Staubli VAL3: HIT_YD.pjx

--- HIT_YD.pjx ---
Parameters version=s7.6.2 stackSize=5000 millimeterUnit=true
Program file=ClientGet.pgx
Program file=ClientSend.pgx
Program file=OMAC_Abort.pgx
Program file=OMAC_Hold.pgx
Program file=OMAC_Main.pgx
Program file=OMAC_Reset.pgx
Program file=OMAC_Start.pgx
Program file=OMAC_Stop.pgx
Program file=OMAC_Unhold.pgx
Program file=blow.pgx
Program file=bypassPick.pgx
Program file=cellManager.pgx
Program file=getToolStatus.pgx
Program file=goHome.pgx
Program file=init.pgx
Program file=initTracking.pgx
Program file=isInSafetyArea.pgx
Program file=modbusGet.pgx
Program file=modbusSet.pgx
Program file=overflowPick.pgx
Program file=Place.pgx
Program file=productionCycle.pgx
Program file=robot2PLC.pgx
Program file=sRobot2fRobot.pgx
Program file=send2NextRob.pgx
Program file=setAlarm.pgx
Program file=setConvSpeed.pgx
Program file=start.pgx
Program file=stop.pgx
Program file=trackErr_init.pgx
Program file=trackingPick.pgx
Program file=transferQueue.pgx
Data file=HIT_YD.dtx
Library alias=mot path=Disk://Tracking/Motion/Motion.pjx autoload=true password=
Type name=object path=Disk://Tracking/Templates/object/object.pjx

--- HIT_YD.dtx ---
aio aConvSpeed = {link=ModbusSrv-0\Modbus-Word\ao[3]}
aio aPlcCmd = {link=ModbusSrv-0\Modbus-Word\ai[0]}
aio aRbAlarm = {link=ModbusSrv-0\Modbus-Word\ao[0]}
aio aRbStatus = {link=ModbusSrv-0\Modbus-Word\ao[1]}
bool _bConvExist = true
bool _bEndCycle
bool _bIsPicking
bool _bIsPlacing
bool _bMutexCnvQueue = true
bool _bPartInTool
bool _bSentToHome = true
bool bIsPermitPlace = true
bool bIsStartPlace = true
bool bLockPage
bool bPickDetection
bool bSetConvSpeed
bool bTransferData
dio dAlarm[8]
  [0] = {link=ModbusSrv-0\Modbus-Bit\do[8]}
  [1] = {link=ModbusSrv-0\Modbus-Bit\do[9]}
  [2] = {link=ModbusSrv-0\Modbus-Bit\do[10]}
  [3] = {link=ModbusSrv-0\Modbus-Bit\do[11]}
  [4] = {link=ModbusSrv-0\Modbus-Bit\do[12]}
  [5] = {link=ModbusSrv-0\Modbus-Bit\do[13]}
  [6] = {link=ModbusSrv-0\Modbus-Bit\do[14]}
  [7] = {link=ModbusSrv-0\Modbus-Bit\do[15]}
dio dBlow = {link=BasicIO-1\%Q5}
dio dControlVacuum[4]
  [0] = {link=BasicIO-1\%Q7}
  [1] = {link=BasicIO-1\%Q6}
  [2] = {link=BasicIO-1\%Q5}
  [3] = {link=BasicIO-1\%Q4}
dio dPartInTool = {link=fIn0}
dio dPermitPlace[4]
  [0] = {link=ModbusSrv-0\Modbus-Bit\di[3]}
  [1] = {link=ModbusSrv-0\Modbus-Bit\di[2]}
  [2] = {link=ModbusSrv-0\Modbus-Bit\di[1]}
  [3] = {link=ModbusSrv-0\Modbus-Bit\di[0]}
dio dPlaceDone[4]
  [0] = {link=ModbusSrv-0\Modbus-Bit\do[3]}
  [1] = {link=ModbusSrv-0\Modbus-Bit\do[2]}
  [2] = {link=ModbusSrv-0\Modbus-Bit\do[1]}
  [3] = {link=ModbusSrv-0\Modbus-Bit\do[0]}
dio dStartControl[4]
  [0] = {link=ModbusSrv-0\Modbus-Bit\di[4]}
  [1] = {link=ModbusSrv-0\Modbus-Bit\di[5]}
  [2] = {link=ModbusSrv-0\Modbus-Bit\di[6]}
  [3] = {link=ModbusSrv-0\Modbus-Bit\di[7]}
dio dStartState[4]
  [0] = {link=ModbusSrv-0\Modbus-Bit\do[4]}
  [1] = {link=ModbusSrv-0\Modbus-Bit\do[5]}
  [2] = {link=ModbusSrv-0\Modbus-Bit\do[6]}
  [3] = {link=ModbusSrv-0\Modbus-Bit\do[7]}
dio dVacuum = {link=BasicIO-1\%Q4}
frame fConveyor = {x=690.465999, y=-334.533545, z=-72.519533, rx=0.736674, ry=-0.299775, rz=179.886741, fatherId=world[0]}
frame fDetection = {x=319.933347, y=-456.969728, z=-77.119399, rx=1.134288, ry=-0.307561, rz=179.705392, fatherId=world[0]}
jointRs jDropPart = {j1=-61.262813, j2=45.342289, j3=74.332986, j4=152.342331}
jointRs jHome = {j1=-61.262813, j2=45.342289, j3=74.332986, j4=152.342331}
jointRs jPark = {j1=-61.262813, j2=45.342289, j3=74.332986, j4=152.342331}
mdesc _mLoad = {accel=64, vel=80, decel=64, leave=30, reach=30}
mdesc mLoad = {accel=64, vel=80, decel=64, leave=30, reach=30}
mdesc mNomSpeed = {accel=144, vel=120, decel=144, leave=20, reach=20}
mdesc mPickDown = {accel=169, vel=130, decel=169, blend=off, leave=30, reach=30}
mdesc mPickup = {accel=144, vel=120, decel=144}
mdesc mPlaceDown = {accel=144, vel=120, decel=144, blend=off, leave=15, reach=15}
mdesc mPlaceUp = {accel=169, vel=130, decel=169, blend=cartesian, leave=30, reach=30}
mdesc mSlow = {accel=1, vel=10, decel=1, leave=10, reach=10}
mdesc mUnload = {accel=121, vel=120, decel=121, leave=40, reach=40}
num _nBlowDelay
num _nCntBypassed
num _nCntPartsDone[2]
  [0] = 13306
  [1] = 13306
num _nCntTransfered = 8
num _nConvSpd = 491.491944
num _nCycleTime[10]
  [0] = 0.964
  [1] = 2.051
  [2] = 0.756
  [3] = 4.461
  [4] = 0.846
  [5] = 4.253
  [6] = 0.92
  [7] = 8.599
  [8] = 0.993
  [9] = 2.124
num _nCycleTimeIndx
num _nID = -1
num _nLastStateCMD
num _nOmacStat = 3
num _nPartID = 1
num _nPlaceCurItem[2]
num _nPullIndexTQ
num _nPushIndexTQ
num _nStateCMD
num _nTimer = 7404.541
num _nTrackErr = 46
num nBlowID = 0.5
num nBypass
num nLoadRatio[4]
  [0] = 1
  [1] = 0.85
  [2] = 0.7
  [3] = 0.7
num nNomConvSpeed = 100
num nPartHeight = 8
num nPickAppro = 60
num nPlaceAppro = 50
num nPlaceCycleNum = 1
public num nPlaceNum = 1
num nSafeMaxX = 850
num nSafeMaxY = 850
num nSafeMinX = -850
num nSafeMinY = -850
num nTestData[5]
  [0] = 1
  [1] = 8
  [3] = -7
num nVacuumID = 0.2
num nWaitDist2Up4BP = -150
num nWaitDistToDown = 50
num nWaitDistToUp[1 3]
  [0,0] = -50
  [0,1] = 200
  [0,2] = 400
num nWaitDistX = -150
object _oTransferQueue[1 100]
  [0,0]
    num nID = -1
    num nLatchedValue
    trsf trTrsf
  [0,1]
    num nID = -1
    num nLatchedValue
    trsf trTrsf
  [0,2]
    num nID = -1
    num nLatchedValue
    trsf trTrsf
  [0,3]
    num nID = -1
    num nLatchedValue
    trsf trTrsf
  [0,4]
    num nID = -1
    num nLatchedValue
    trsf trTrsf
  [0,5]
    num nID = -1
    num nLatchedValue
    trsf trTrsf
  [0,6]
    num nID = -1
    num nLatchedValue
    trsf trTrsf
  [0,7]
    num nID = -1
    num nLatchedValue
    trsf trTrsf
  [0,8]
    num nID = -1
    num nLatchedValue
    trsf trTrsf
  [0,9]
    num nID = -1
    num nLatchedValue
    trsf trTrsf
  [0,10]
    num nID = -1
    num nLatchedValue
    trsf trTrsf
  [0,11]
    num nID = -1
    num nLatchedValue
    trsf trTrsf
  [0,12]
    num nID = -1
    num nLatchedValue
    trsf trTrsf
  [0,13]
    num nID = -1
    num nLatchedValue
    trsf trTrsf
  [0,14]
    num nID = -1
    num nLatchedValue
    trsf trTrsf
  [0,15]
    num nID = -1
    num nLatchedValue
    trsf trTrsf
  [0,16]
    num nID = -1
    num nLatchedValue
    trsf trTrsf
  [0,17]
    num nID = -1
    num nLatchedValue
    trsf trTrsf
  [0,18]
    num nID = -1
    num nLatchedValue
    trsf trTrsf
  [0,19]
    num nID = -1
    num nLatchedValue
    trsf trTrsf
  [0,20]
    num nID = -1
    num nLatchedValue
    trsf trTrsf
  [0,21]
    num nID = -1
    num nLatchedValue
    trsf trTrsf
  [0,22]
    num nID = -1
    num nLatchedValue
    trsf trTrsf
  [0,23]
    num nID = -1
    num nLatchedValue
    trsf trTrsf
  [0,24]
    num nID = -1
    num nLatchedValue
    trsf trTrsf
  [0,25]
    num nID = -1
    num nLatchedValue
    trsf trTrsf
  [0,26]
    num nID = -1
    num nLatchedValue
    trsf trTrsf
  [0,27]
    num nID = -1
    num nLatchedValue
    trsf trTrsf
  [0,28]
    num nID = -1
    num nLatchedValue
    trsf trTrsf
  [0,29]
    num nID = -1
    num nLatchedValue
    trsf trTrsf
  [0,30]
    num nID = -1
    num nLatchedValue
    trsf trTrsf
  [0,31]
    num nID = -1
    num nLatchedValue
    trsf trTrsf
  [0,32]
    num nID = -1
    num nLatchedValue
    trsf trTrsf
  [0,33]
    num nID = -1
    num nLatchedValue
    trsf trTrsf
  [0,34]
    num nID = -1
    num nLatchedValue
    trsf trTrsf
  [0,35]
    num nID = -1
    num nLatchedValue
    trsf trTrsf
  [0,36]
    num nID = -1
    num nLatchedValue
    trsf trTrsf
  [0,37]
    num nID = -1
    num nLatchedValue
    trsf trTrsf
  [0,38]
    num nID = -1
    num nLatchedValue
    trsf trTrsf
  [0,39]
    num nID = -1
    num nLatchedValue
    trsf trTrsf
  [0,40]
    num nID = -1
    num nLatchedValue
    trsf trTrsf
  [0,41]
    num nID = -1
    num nLatchedValue
    trsf trTrsf
  [0,42]
    num nID = -1
    num nLatchedValue
    trsf trTrsf
  [0,43]
    num nID = -1
    num nLatchedValue
    trsf trTrsf
  [0,44]
    num nID = -1
    num nLatchedValue
    trsf trTrsf
  [0,45]
    num nID = -1
    num nLatchedValue
    trsf trTrsf
  [0,46]
    num nID = -1
    num nLatchedValue
    trsf trTrsf
  [0,47]
    num nID = -1
    num nLatchedValue
    trsf trTrsf
  [0,48]
    num nID = -1
    num nLatchedValue
    trsf trTrsf
  [0,49]
    num nID = -1
    num nLatchedValue
    trsf trTrsf
  [0,50]
    num nID = -1
    num nLatchedValue
    trsf trTrsf
  [0,51]
    num nID = -1
    num nLatchedValue
    trsf trTrsf
  [0,52]
    num nID = -1
    num nLatchedValue
    trsf trTrsf
  [0,53]
    num nID = -1
    num nLatchedValue
    trsf trTrsf
  [0,54]
    num nID = -1
    num nLatchedValue
    trsf trTrsf
  [0,55]
    num nID = -1
    num nLatchedValue
    trsf trTrsf
  [0,56]
    num nID = -1
    num nLatchedValue
    trsf trTrsf
  [0,57]
    num nID = -1
    num nLatchedValue
    trsf trTrsf
  [0,58]
    num nID = -1
    num nLatchedValue
    trsf trTrsf
  [0,59]
    num nID = -1
    num nLatchedValue
    trsf trTrsf
  [0,60]
    num nID = -1
    num nLatchedValue
    trsf trTrsf
  [0,61]
    num nID = -1
    num nLatchedValue
    trsf trTrsf
  [0,62]
    num nID = -1
    num nLatchedValue
    trsf trTrsf
  [0,63]
    num nID = -1
    num nLatchedValue
    trsf trTrsf
  [0,64]
    num nID = -1
    num nLatchedValue
    trsf trTrsf
  [0,65]
    num nID = -1
    num nLatchedValue
    trsf trTrsf
  [0,66]
    num nID = -1
    num nLatchedValue
    trsf trTrsf
  [0,67]
    num nID = -1
    num nLatchedValue
    trsf trTrsf
  [0,68]
    num nID = -1
    num nLatchedValue
    trsf trTrsf
  [0,69]
    num nID = -1
    num nLatchedValue
    trsf trTrsf
  [0,70]
    num nID = -1
    num nLatchedValue
    trsf trTrsf
  [0,71]
    num nID = -1
    num nLatchedValue
    trsf trTrsf
  [0,72]
    num nID = -1
    num nLatchedValue
    trsf trTrsf
  [0,73]
    num nID = -1
    num nLatchedValue
    trsf trTrsf
  [0,74]
    num nID = -1
    num nLatchedValue
    trsf trTrsf
  [0,75]
    num nID = -1
    num nLatchedValue
    trsf trTrsf
  [0,76]
    num nID = -1
    num nLatchedValue
    trsf trTrsf
  [0,77]
    num nID = -1
    num nLatchedValue
    trsf trTrsf
  [0,78]
    num nID = -1
    num nLatchedValue
    trsf trTrsf
  [0,79]
    num nID = -1
    num nLatchedValue
    trsf trTrsf
  [0,80]
    num nID = -1
    num nLatchedValue
    trsf trTrsf
  [0,81]
    num nID = -1
    num nLatchedValue
    trsf trTrsf
  [0,82]
    num nID = -1
    num nLatchedValue
    trsf trTrsf
  [0,83]
    num nID = -1
    num nLatchedValue
    trsf trTrsf
  [0,84]
    num nID = -1
    num nLatchedValue
    trsf trTrsf
  [0,85]
    num nID = -1
    num nLatchedValue
    trsf trTrsf
  [0,86]
    num nID = -1
    num nLatchedValue
    trsf trTrsf
  [0,87]
    num nID = -1
    num nLatchedValue
    trsf trTrsf
  [0,88]
    num nID = -1
    num nLatchedValue
    trsf trTrsf
  [0,89]
    num nID = -1
    num nLatchedValue
    trsf trTrsf
  [0,90]
    num nID = -1
    num nLatchedValue
    trsf trTrsf
  [0,91]
    num nID = -1
    num nLatchedValue
    trsf trTrsf
  [0,92]
    num nID = -1
    num nLatchedValue
    trsf trTrsf
  [0,93]
    num nID = -1
    num nLatchedValue
    trsf trTrsf
  [0,94]
    num nID = -1
    num nLatchedValue
    trsf trTrsf
  [0,95]
    num nID = -1
    num nLatchedValue
    trsf trTrsf
  [0,96]
    num nID = -1
    num nLatchedValue
    trsf trTrsf
  [0,97]
    num nID = -1
    num nLatchedValue
    trsf trTrsf
  [0,98]
    num nID = -1
    num nLatchedValue
    trsf trTrsf
  [0,99]
    num nID = -1
    num nLatchedValue
    trsf trTrsf
pointRs pPick = {shoulder=righty, fatherId=fDetection[0]}
pointRs pPlace[4]
  [0] = {x=752.590073, y=-120.83, z=-69.15, rx=180, rz=95.410382, shoulder=righty, fatherId=world[0]}
  [1] = {x=614.985623, y=-120.83, z=-69.15, rx=180, rz=95.41037, shoulder=righty, fatherId=world[0]}
  [2] = {x=479.250185, y=-120.83, z=-69.15, rx=180, rz=95.410122, shoulder=righty, fatherId=world[0]}
  [3] = {x=345.150595, y=-120.83, z=-69.15, rx=180, rz=95.409269, shoulder=righty, fatherId=world[0]}
sio sClient = {link=Socket\StlClient}
sio skToRobot = {link=Socket\toRobot_sk1}
string _sCycleStatus = "Waiting for part to pick"
string sConveyorList = "cvIn"
string sSecondRStatus = "8"
tool tGripper = {z=75, rz=-128, fatherId=flange[0], ioLink=valve1}
public trsf trTrsfPlace[4]
  [1] = {x=140}
  [2] = {x=280}
  [3] = {x=420}

--- cellManager.pgx ---
program cellManager()
  local joint l_jHere
  local num l_nConvSpeedOld
  local num l_nErr
  local num l_nI
begin
  // This program is the cell manager, it manage:
  //  -  Variable initializing
  //  -  Launch Tracking
  //  -  Arm Power
  //  -  Robot home position
  //  -  Launch user’s tasks, kills and re-launch user’s task in case of tracking error
  //  -  Displays cycle times and counters.
  //
  // Input parameters
  //  None            :
  //
  // Output parameters
  //  None            :
  //
  //----------------------------------------------------------------
  //

  //  //Launch queue transfer tasks
  //  if _bTransferData[0]
  //    taskCreate "TransferQueue1",100,transferQueue(0)
  //  endIf
  //  // Task to remove picking positions that have pass the downstream limit while the robot is placing a part.
  //  taskCreate "overflowPick",100,overflowPick()

  // Task for production cycle
  if taskStatus("productionCycle")>=0
    taskKill("productionCycle")
  endIf
  wait(taskStatus("productionCycle")<0)
  taskCreate "productionCycle",100,productionCycle()


  // Task to set the blow on the tool for a defined period of time
  if taskStatus("blow")>=0
    taskKill("blow")
  endIf
  wait(taskStatus("blow")<0)
  taskCreate "blow",100,blow()
  wait(taskStatus("blow")==1)
  //
  if taskStatus("sRobot2fRobot")>=0
    taskKill("sRobot2fRobot")
  endIf
  wait(taskStatus("sRobot2fRobot")<0)
  taskCreate "sRobot2fRobot",100,sRobot2fRobot()
  //
  if taskStatus("robot2PLC")>=0
    taskKill("robot2PLC")
  endIf
  wait(taskStatus("robot2PLC")<0)
  taskCreate "robot2PLC",100,robot2PLC()

  //OMAC进程:Running
  _nOmacStat=3

  //
  //  //Init conveyor speed
  //  call setConvSpeed(0,nNomConvSpeed[0])
  //  l_nConvSpeedOld[0]=nNomConvSpeed[0]
  //
  // Main loop
  do
    // Enable Power
    if isPowered()==false and esStatus()!=2
      if _nOmacStat==3
        enablePower()
        delay(0.5)
      endIf
    endIf
    //
    // Set conveyor speed to the nominal value if the conveyor speed is not controlled by the tasks
    //  overflowPick and overflowPlace
    if bSetConvSpeed[0]
      l_nConvSpeedOld[0]=0
    else
      if l_nConvSpeedOld[0]!=nNomConvSpeed[0]
        call setConvSpeed(0,nNomConvSpeed[0])
        l_nConvSpeedOld[0]=nNomConvSpeed[0]
      endIf
    endIf

    if _nOmacStat==3
      //task TransferQueue1 error management,auto recover
      if bTransferData[0]
        if taskStatus("TransferQueue1")!=1
          logMsg("TransferQueue1任务错误")
          taskKill("TransferQueue1")
          wait(taskStatus("TransferQueue1")==-1)
          taskCreate "TransferQueue1",100,transferQueue(0)
          wait(taskStatus("TransferQueue1")==1)
          logMsg("TransferQueue1自动恢复")
        endIf
      endIf
      //task TransferQueue1 error management,auto recover
      if taskStatus("overflowPick")!=1
        logMsg("overflowPick任务错误")
        taskKill("overflowPick")
        wait(taskStatus("overflowPick")==-1)
        taskCreate "overflowPick",100,overflowPick()
        wait(taskStatus("overflowPick")==1)
        logMsg("overflowPick自动恢复")
      endIf
      // Tracking error management
      if isSettled()==true and $trackingState()==-1
        if _nOmacStat==3
          if _bIsPicking==true
            logMsg("抓取时跟踪错误")
          endIf
          if _bIsPlacing==true
            logMsg("放件时运动错误")
          endIf
          //记录跟踪错误次数
          _nTrackErr=_nTrackErr+1
          stopMove()
          resetMotion()
          call trackErr_init()
          autoConnectMove(true)
          l_jHere=herej()
          l_jHere.j3=jHome.j3
          movej(l_jHere,tGripper,mNomSpeed)
          movej(jHome,tGripper,mNomSpeed)
          _bSentToHome=true
          //          //Launch queue transfer tasks
          //          if _bTransferData[0]
          //            taskCreate "TransferQueue1",100,transferQueue(0)
          //          endIf
          //          // Task to remove picking positions that have pass the downstream limit while the robot is placing a part.
          //          taskCreate "overflowPick",100,overflowPick()
          // Task for production cycle

          if taskStatus("productionCycle")>=0
            taskKill("productionCycle")
          endIf
          wait(taskStatus("productionCycle")<0)
          taskCreate "productionCycle",100,productionCycle()
          wait(taskStatus("productionCycle")==1)
        endIf
      endIf
    endIf
    //
    //show cv speed
    if _bConvExist
      call mot:getConvSpeed(0,_nConvSpd,l_nErr)
      gotoxy(0,0)
      put("                    ")
      gotoxy(0,0)
      put("传送带速度："+toString("",_nConvSpd)+" mm/s")
    endIf


    delay(0)
  until false
end

--- init.pgx ---
program init()
  local num l_nI
  local num l_nJ
begin
  // This program initialize all variables
  //
  // Input parameters
  //  None            :
  //
  // Output parameters
  //  None            :
  //
  //----------------------------------------------------------------
  //
  //che add
  nPlaceNum=0
  nPlaceCycleNum=0
  bIsPermitPlace=true
  sSecondRStatus=""
  // Booleans
  _bSentToHome=false
  _bMutexCnvQueue[0]=false
  _bIsPicking=false
  _bIsPlacing=false
  _bConvExist=false
  _bEndCycle=false
  //

  //
  // Numerical
  _nBlowDelay=0
  _nID[0]=-1
  _nCntBypassed[0]=nBypass[0]
  _nCntTransfered[0]=0

  _nPushIndexTQ[0]=0
  _nPullIndexTQ[0]=0
  _nTimer=0

  resize(_nCycleTime,1,10)
  for _nCycleTimeIndx=0 to size(_nCycleTime)-1
    _nCycleTime[_nCycleTimeIndx]=0
  endFor
  _nCycleTimeIndx=0

  //dio
  dPlaceDone[0]=false
  dPlaceDone[1]=false
  dPlaceDone[2]=false
  dPlaceDone[3]=false

  // aio
  aioSet(aRbAlarm,0)
  //call setAlarm(0)

  //
  // Points
  pPick.trsf={0,0,0,0,0,0}

  //

  //
  // Transfer Queues
  for l_nI=0 to size(_oTransferQueue,2)-1
    _oTransferQueue[0,l_nI].nID=-1
    _oTransferQueue[0,l_nI].trTrsf={0,0,0,0,0,0}
    _oTransferQueue[0,l_nI].nLatchedValue=0
  endFor
  //
  // Strings
  _sCycleStatus=""
end

--- isInSafetyArea.pgx ---
program isInSafetyArea()
  local jointRs l_jHere
  local pointRs l_pCurrent
begin
  do
    l_pCurrent=here(flange,world)
    //**************************************************//
    //******** 用来判断机器人是否在安全工作空间 ********//
    //**************************************************//
    if (l_pCurrent.trsf.y>=nSafeMaxY or l_pCurrent.trsf.y<=nSafeMinY or l_pCurrent.trsf.x>=nSafeMaxX or l_pCurrent.trsf.x<=nSafeMinX) and _nOmacStat==3
      aioSet(aRbAlarm,10)
      call setAlarm(7)
      popUpMsg("机器人超出安全工作空间！")
      logMsg("机器人超出安全工作空间！")
      call OMAC_Abort()
    endIf
    delay(0)
  until false
end

--- OMAC_Main.pgx ---
program OMAC_Main()
begin
  //  _nOmacStat
  //1-Ready
  //2-Starting
  //3-Running
  //4-Resetting
  //5-Holding
  //6-Held
  //7-Un-Holding
  //8-Stopping
  //9-Stopped
  //10-Aborting


  // _nStateCmd
  //1-Start
  //2-Stop
  //3-Reset
  //4-Hold
  //10-Abort

  //机器人状态
  _nOmacStat=9

  _nLastStateCMD=0
  //OMAC_init
  call init()
  do
    switch _nOmacStat
      //复位信号
      case 1
        call modbusSet(3)
      break
      //运行信号
      case 3
        call modbusSet(1)
      break
      //准备信号
      case 4
        call modbusSet(2)
      break
      //停止信号
      case 9
        call modbusSet(2)
      break
    endSwitch
    //机器人状态输出
    //aioSet(aRbStatus,_nOmacStat)
    //根据上位机按钮转换为指令num
    //10-Abort
    if esStatus()==2
      _nStateCMD=10
    else
      call modbusGet(_nStateCMD)

      //_nStateCMD=aioGet(aPlcCmd)
    endIf

    //根据指令num，触发相应动作
    if _nStateCMD!=_nLastStateCMD
      switch _nStateCMD
        //Reset
        case 3
          //确认当前OMAC进程为stopped
          if _nOmacStat==9

            if taskStatus("Reset")>=0
              taskKill("Reset")
            endIf
            wait(taskStatus("Reset")<0)
            taskCreate "Reset",100,OMAC_Reset()

          endIf
        break

        //Start
        case 1
          //确认当前OMAC进程为Ready
          if _nOmacStat==1

            if taskStatus("Start")>=0
              taskKill("Start")
            endIf
            wait(taskStatus("Start")<0)
            taskCreate "Start",100,OMAC_Start()


          elseIf _nOmacStat==6
            //确认当前OMAC进程为Held

            if taskStatus("Unhold")>=0
              taskKill("Unhold")
            endIf
            wait(taskStatus("Unhold")<0)
            taskCreate "Unhold",100,OMAC_Unhold()

          endIf
        break
        //Hold
        case 4
          //确认当前OMAC进程为running
          if _nOmacStat==3

            if taskStatus("Hold")>=0
              taskKill("Hold")
            endIf
            wait(taskStatus("Hold")<0)
            taskCreate "Hold",100,OMAC_Hold()

          endIf
        break

        //Unhold
        case 7

        break

        //Stop
        case 2
          //确认当前OMAC进程不是停止
          if _nOmacStat!=9
            if taskStatus("Stop")>=0
              taskKill("Stop")
            endIf
            wait(taskStatus("Stop")<0)
            taskCreate "Stop",100,OMAC_Stop()
          endIf
        break

        //Abort
        case 10
          // //确认当前OMAC进程不是停止
          if _nOmacStat!=9
            if taskStatus("Abort")>=0
              taskKill("Abort")
            endIf
            wait(taskStatus("Abort")<0)
            taskCreate "Abort",100,OMAC_Abort()
          endIf
        break

      endSwitch
    endIf
    //记录上次指令
    _nLastStateCMD=_nStateCMD
    delay(0)
  until false


end

--- OMAC_Stop.pgx ---
program OMAC_Stop()
  local joint l_jHere
  local string l_sToolStatus
begin

  //OMAC进程:Stopping
  _nOmacStat=8
  logMsg("上位机手动操作：停止")
  stopMove()
  resetMotion()
  //
  // Stop task

  taskKill("cellManager")
  taskKill("overflowPick")
  taskKill("productionCycle")
  taskKill("Reset")
  taskKill("Start")
  taskKill("Hold")
  taskKill("Unhold")
  taskKill("Preheat")
  taskKill("openPallet")
  taskKill("changeBox")
  taskKill("convStopCheck")
  taskKill("TransferQueue1")
  taskKill("robot2PLC")
  taskKill("sRobot2fRobot")


  resetMotion()
  while !isPowered()
    enablePower()
    delay(1)
  endWhile
  //
  // Move up axis 3
  l_jHere=herej()
  l_jHere.j3=95
  movej(l_jHere,tGripper,mSlow)
  //
  // Drop the part on the tool
  if bPickDetection==true
    call getToolStatus(l_sToolStatus)
  endIf
  if l_sToolStatus=="PartInTool" or !bPickDetection
    movej(jDropPart,tGripper,mSlow)
    waitEndMove()
    dVacuum=false
  else
    dVacuum=false
  endIf
  //
  // Go to park position
  movej(jPark,tGripper,mSlow)
  waitEndMove()
  wait(taskStatus("Reset")==-1)
  wait(taskStatus("Start")==-1)
  wait(taskStatus("Hold")==-1)
  wait(taskStatus("Unhold")==-1)
  wait(taskStatus("Preheat")==-1)
  wait(taskStatus("openPallet")==-1)
  wait(taskStatus("changeBox")==-1)
  wait(taskStatus("convStopCheck")==-1)
  wait(taskStatus("cellManager")==-1)
  wait(taskStatus("TransferQueue1")==-1)
  wait(taskStatus("overflowPick")==-1)
  wait(taskStatus("productionCycle")==-1)

  if _bConvExist
    call mot:kill()
    _bConvExist=false
  endIf

  disablePower()
  wait(isPowered()==false)
  //OMAC进程:Stopped
  _nOmacStat=9

  delay(0)
end

--- Place.pgx ---
program place()
  local bool l_bNoError
  local joint l_jAppro
  local num l_nConvNum
  local num l_nError
  local num l_nMoveID
  local num l_nTrackStatus
  local pointRs l_pAppro
  local pointRs l_pPlace
  local string l_sToolStatus
begin
  l_nConvNum=1
  link(l_pPlace,world)
  //che modify start
  if nPlaceNum>3
    nPlaceNum=0
  endIf
  _mLoad=mLoad
  _mLoad.vel=mLoad.vel*nLoadRatio[nPlaceNum]
  _mLoad.accel=mLoad.accel*nLoadRatio[nPlaceNum]*nLoadRatio[nPlaceNum]
  _mLoad.decel=mLoad.decel*nLoadRatio[nPlaceNum]*nLoadRatio[nPlaceNum]
  if nPlaceCycleNum>7
    nPlaceCycleNum=0
  endIf

  //dControlVacuum[nPlaceNum]=false
  l_pPlace=pPlace[nPlaceNum]
  //end
  // Place part
  l_pAppro=appro(l_pPlace,{0,0,-nPlaceAppro,0,0,0})
  l_bNoError=pointToJoint(tGripper,jHome,l_pAppro,l_jAppro)
  call mot:getTrackStatus(l_nTrackStatus)
  if l_nTrackStatus>0
    // Use trackOff if the robot is synchronized
    if l_bNoError
      call mot:trackOffJ(l_jAppro,tGripper,_mLoad,l_nMoveID,l_nError)
    else
      call mot:trackOff(l_pAppro,tGripper,_mLoad,l_nMoveID,l_nError)
    endIf
  else
    // Use movej if the robot is not synchronized
    if l_bNoError
      l_nMoveID=movej(l_jAppro,tGripper,_mLoad)
    else
      l_nMoveID=movej(l_pAppro,tGripper,_mLoad)
    endIf
  endIf
  // wait permit signal
  wait(bIsPermitPlace==true)
  wait(dPermitPlace[nPlaceNum]==true)
  movel(l_pPlace,tGripper,mPlaceDown)
  l_nMoveID=movel(l_pAppro,tGripper,mPlaceUp)
  // check PartInTool if bPickDetection
  if bPickDetection
    //wait(getMoveId()>l_nMoveID-0.8)
    wait(getMoveId()>l_nMoveID+nBlowID-1.1)
    call getToolStatus(l_sToolStatus)
  else
    wait(getMoveId()>l_nMoveID+nBlowID-1.1)
    _bPartInTool=false
  endIf
  //Blow
  wait(getMoveId()>l_nMoveID+nBlowID-1)
  _nBlowDelay=0.15
  // send done signal
  //dPlaceDone[nPlaceNum]=true
  wait(getMoveId()>l_nMoveID+0.1)
  delay(0)
  //dPlaceDone[nPlaceNum]=false
  if l_sToolStatus=="PartInTool" or _bPartInTool==false
    // A part has been placed
    _nCntPartsDone[l_nConvNum]=_nCntPartsDone[l_nConvNum]+1
  endIf
  delay(0)
  //che modify start
  delay(0)

  //sClient=toString("",nPlaceCycleNum)
  nPlaceCycleNum=nPlaceCycleNum+1
  nPlaceNum=nPlaceNum+1
  dPlaceDone[nPlaceNum-1]=true
  //end

end

--- productionCycle.pgx ---
program productionCycle()
  local bool l_bPartDone
  local string l_sToolStatus
begin
  // This program is the main cycle. It pick on part from the input
  // conveyor and places it on an empty cavity on the output conveyor.
  //
  // Input parameters
  //  None            :
  //
  // Output parameters
  //  None            :
  //
  //----------------------------------------------------------------
  //
  // In order to improve cycle time, vacuum is always on, even while
  //  placing a part. To place a part, the blow is activated for a
  //  short period of time when the robot arrives to the place position.
  //
  // Main loop

  call getToolStatus(l_sToolStatus)
  if (!bPickDetection and _bPartInTool==true) or (bPickDetection and l_sToolStatus=="PartInTool")
    call place()
  endIf
  //---------------------------------------------------------------------//
  do
    //Takes control of the Pick conveyor queue.
    setMutex(_bMutexCnvQueue[0])
    do
      call trackingPick(l_bPartDone)
      delay(0)
    until l_bPartDone
    // Release control of the Pick conveyor queue.
    _bMutexCnvQueue[0]=false

    //
    call place()
    //
    delay(0)
  until _bEndCycle
  _bEndCycle=true
  //
end

--- robot2PLC.pgx ---
program robot2PLC()
  local num l_nLocalNum
  local num l_nNextNum
  local num l_ns
begin
  l_nLocalNum=-1
  while true
    //

    wait(dPlaceDone[0]==true or dPlaceDone[1]==true or dPlaceDone[2]==true or dPlaceDone[3]==true)
    //
    l_ns=clock()
    do
      delay(0)
    until clock()-l_ns>0.25

    if (dPlaceDone[0]==true)
      dPlaceDone[0]=false
    elseIf (dPlaceDone[1]==true)
      dPlaceDone[1]=false
    elseIf (dPlaceDone[2]==true)
      dPlaceDone[2]=false
    elseIf (dPlaceDone[3]==true)
      dPlaceDone[3]=false
    else
      dPlaceDone[0]=false
      dPlaceDone[1]=false
      dPlaceDone[2]=false
      dPlaceDone[3]=false
    endIf
    //
    sClient=toString("",nPlaceCycleNum)
    //    if (l_nLocalNum!=nPlaceCycleNum)
    //      //
    //      sClient=toString("",nPlaceCycleNum)
    //      l_nLocalNum=nPlaceCycleNum
    //    endIf

    nTestData[0]=nPlaceCycleNum
    nTestData[1]=asc(sSecondRStatus,0)-48
    nTestData[3]=nTestData[0]-nTestData[1]
  endWhile
end

--- sRobot2fRobot.pgx ---
program sRobot2fRobot()
begin

  //没有ClearBuffer 这个比较难联通
  clearBuffer(sClient)

  //把客户端收到不为空的信息通过服务器传送出去
  while true
    //服务器
    //clearBuffer(sServer)

    call ClientGet(sSecondRStatus)
    //popUpMsg(sFirstRStatus)

    delay(0)
  endWhile

end

--- stop.pgx ---
program stop()
  local joint l_jHere
  local string l_sToolStatus
begin
  //
  l_sToolStatus=""
  //
  cls()
  gotoxy(10,6)
  put("Application Ending")
  //
  stopMove()
  resetMotion()
  disablePower()
  // Stop all tasks
  taskKill("TransferQueue1")
  taskKill("overflowPick")
  taskKill("productionCycle")
  taskKill("blow")
  taskKill("changePallet")
  taskKill("isInSafetyArea")
  taskKill("robot2PLC")
  taskKill("sRobot2fRobot")

  if _bConvExist
    call mot:kill()
  endIf

  //
  // Stop conveyor speed
  call setConvSpeed(0,0)
  //
  // Reset triggers
  //  dioSet(dTrigger,0)
  //
  resetMotion()
  //
  //
  // Move up axis 3
  l_jHere=herej()
  l_jHere.j3=90
  //movej(l_jHere,flange,mSlow)
  //
  // Drop the part on the tool
  if bPickDetection
    call getToolStatus(l_sToolStatus)
  endIf
  if l_sToolStatus=="PartInTool" or !bPickDetection
    //movej(jDropPart,flange,mSlow)
    //waitEndMove()
    dBlow=true
    dVacuum=false
    delay(0.5)
    dBlow=false
  else
    dVacuum=false
    dBlow=false
  endIf
  //
  // Go to park position
  //movej(jPark,flange,mSlow)
  //waitEndMove()
  disablePower()
  //
  cls()
  gotoxy(10,6)
  put("Application Ended")
  //
end

--- trackErr_init.pgx ---
program trackErr_init()
  local num l_nI
begin
  // This program initialize all variables
  //
  // Input parameters
  //  None            :
  //
  // Output parameters
  //  None            :
  //
  //----------------------------------------------------------------
  //
  // Booleans
  _bSentToHome=false
  _bMutexCnvQueue[0]=false
  _bIsPicking=false
  _bIsPlacing=false
  //

  //
  // Numerical
  _nID[0]=-1
  _nCntBypassed[0]=nBypass[0]


  _nPushIndexTQ[0]=0
  _nPullIndexTQ[0]=0
  _nTimer=0

  for _nCycleTimeIndx=0 to 9
    _nCycleTime[_nCycleTimeIndx]=0
  endFor
  _nCycleTimeIndx=0
  //
  // Points
  pPick.trsf={0,0,0,0,0,0}

  //
  // Transfer Queues
  for l_nI=0 to size(_oTransferQueue,2)-1
    _oTransferQueue[0,l_nI].nID=-1
    _oTransferQueue[0,l_nI].trTrsf={0,0,0,0,0,0}
    _oTransferQueue[0,l_nI].nLatchedValue=0
  endFor
  //
  // Strings
  _sCycleStatus=""
end

--- trackingPick.pgx ---
program trackingPick(bool& x_bPartDone (dimensions=1))
  local bool l_bNoError
  local bool l_bSent2WaitPos
  local joint l_jAppro
  local num l_nConvNum
  local num l_nDistToDown
  local num l_nDistToUp
  local num l_nEncLatchVal
  local num l_nError
  local num l_nMoveID
  local num l_nTrackOnID
  local num l_nTrackStatus
  local point l_pAppro
  local string l_sToolStatus
begin
  // This program picks a part from the input conveyor.
  // If there isn’t an object on the conveyor’s queue, the robot
  //  moves to the home position and waits until there is an object
  //  on the conveyor’s queue.
  // If there is an object on the conveyor’s queue but the object is
  //  upstream of the upstream limit, the robot moves above the
  //  conveyor aligned in front of the object and waits until the
  //  object crosses the upstream limit.
  // If the object is in between the upstream and downstream limit,
  //  the robot picks the part.
  // If the object is downstream of the downstream limit, the object
  //  is removed from the conveyor’s queue and the robot is sent to
  //  the home position.
  //
  // Input parameters
  //  None            :
  //
  // Output parameters
  //  x_bPartDone     : A part has been picked
  //
  //----------------------------------------------------------------
  //
  l_nConvNum=0
  x_bPartDone=false
  l_sToolStatus=""
  //
  // If the overflowPick task hasn't already detect the next part to pick,
  //  wait until an object is present in the queue
  _sCycleStatus="Waiting for part to pick"
  while (_nID[l_nConvNum]==-1)
    call mot:getNextID(l_nConvNum,_nID[l_nConvNum])
    // Send the robot to home if there isn’t a part available and if the robot hasn’t been sent to home.
    if _nID[l_nConvNum]==-1 and !_bSentToHome
      call goHome(l_nMoveID)
    endIf
    delay(0)
  endWhile
  _bIsPicking=true
  _nPartID=_nID[l_nConvNum]
  //
  // If the overflowPick task hasn't already detect the next part to pick,
  //  recover next point transformation from the stack
  if pPick.trsf=={0,0,0,0,0,0}
    call mot:getObjectData(l_nConvNum,pPick.trsf,l_nError)
  endIf
  pPick.trsf.z=nPartHeight
  //若视觉发送的y坐标小于-90，停机、报警
  if pPick.trsf.y<-100
    aioSet(aRbAlarm,50)
    call setAlarm(4)
    stopMove()
    resetMotion()
    disablePower()
    popUpMsg("物件y坐标错误: y="+toString("0.2",pPick.trsf.y))
    logMsg("物件y坐标错误: y="+toString("0.2",pPick.trsf.y))
    call OMAC_Abort()
  endIf
  //
  // If the object is upstream of the upstream limit, send the robot to a
  //  waiting position above the conveyor aligned in front of the object and
  //  waits until the part crosses the upstream limit.
  l_bSent2WaitPos=false
  do
    call mot:getDistance(l_nConvNum,pPick,0,l_nDistToUp,l_nDistToDown,l_nError)
    _sCycleStatus="Distance to pick: "+toString("7.2",l_nDistToUp)
    if l_nDistToUp<nWaitDistToUp[l_nConvNum,0] and !l_bSent2WaitPos
      //
      l_bSent2WaitPos=true
      //
      // Compute waiting position
      l_pAppro=appro(pPick,{0,0,nPickAppro,180,0,0})
      l_pAppro.trsf.x=nWaitDistToUp[0,0]+nWaitDistX
      l_bNoError=pointToJoint(tGripper,jHome,l_pAppro,l_jAppro)
      //
      // Move to the waiting position
      call mot:getTrackStatus(l_nTrackStatus)
      if l_nTrackStatus>0
        // Use trackOff if the robot is synchronized
        if l_bNoError
          call mot:trackOffJ(l_jAppro,tGripper,mUnload,l_nMoveID,l_nError)
        else
          call mot:trackOff(l_pAppro,tGripper,mUnload,l_nMoveID,l_nError)
        endIf
      else
        // Use movej if the robot is not synchronized
        if l_bNoError
          l_nMoveID=movej(l_jAppro,tGripper,mNomSpeed)
        else
          l_nMoveID=movej(l_pAppro,tGripper,mNomSpeed)
        endIf
      endIf
      //
    endIf
    delay(0)
  until (l_nDistToUp>=nWaitDistToUp[l_nConvNum,0])
  //
  // Send the robot to pick the part if the part hasn’t cross the downstream limit,
  //  otherwise remove the part and send the robot to the home position.
  if (l_nDistToUp<nWaitDistToUp[l_nConvNum,1] and !bSetConvSpeed[l_nConvNum]) or (l_nDistToDown<nWaitDistToDown[l_nConvNum] and bSetConvSpeed[l_nConvNum])
    //
    _bSentToHome=false
    //
    // Turn the Z of the point upside down
    pPick=appro(pPick,{0,0,0,180,0,0})
    //
    // Compute approach location
    l_pAppro=appro(pPick,{0,0,-nPickAppro,0,0,0})
    //
    // Move to the part
    if l_bSent2WaitPos
      call mot:trackOn(l_nConvNum,l_pAppro,tGripper,mNomSpeed,l_nTrackOnID,l_nError)
    else
      call mot:trackOnJ(l_nConvNum,l_pAppro,tGripper,jHome,mUnload,l_nTrackOnID,l_nError)
    endIf

    // vacuum
    wait(getMoveId()>l_nTrackOnID+nVacuumID)
    dBlow=false
    dVacuum=true
    call mot:trackOn(l_nConvNum,pPick,tGripper,mPickDown,l_nMoveID,l_nError)
    //    waitEndMove()
    // Compute depart location
    l_pAppro=appro(pPick,{0,0,-nPickAppro,0,0,0})
    //
    // Move up
    call mot:trackOn(l_nConvNum,l_pAppro,tGripper,mPickup,l_nMoveID,l_nError)
    //
    // Wait for the robot to get slightly away from the picking point
    //  and check if the part was taken
    if bPickDetection
      wait(getMoveId()>l_nMoveID+0.5)
      call getToolStatus(l_sToolStatus)
    else
      // Wait until the robot is synchronized with the conveyor to
      //  avoid that the next place routine is executed before the
      //  movements of this pick routine are started.
      wait(getMoveId()>l_nMoveID-0.3)
      _bPartInTool=true
    endIf

    // Remove object from conveyor's queue
    call mot:removePart(l_nConvNum)
    //
    // A part has been picked
    x_bPartDone=true
    _nCntPartsDone[l_nConvNum]=_nCntPartsDone[l_nConvNum]+1
    //
    // Measure Cycle Time
    if _nTimer!=0
      _nCycleTime[_nCycleTimeIndx]=clock()-_nTimer
      _nCycleTimeIndx=(_nCycleTimeIndx+1)%size(_nCycleTime)
      gotoxy(1,0)
      put("                    ")
      gotoxy(1,0)
      put("CT："+toString("",_nCycleTime[_nCycleTimeIndx])+" s")
    endIf
    //
    _nTimer=clock()
    //
    // Reset bypass counter
    _nCntBypassed[l_nConvNum]=0
    //

    //
  else
    // Send the robot to home if the robot hasn’t been sent to home.
    if !_bSentToHome
      call goHome(l_nMoveID)
    endIf
    //
    // Send part to the next robot
    if bTransferData[l_nConvNum]
      call mot:getObjectLatch(l_nConvNum,l_nEncLatchVal,l_nError)
      call send2NextRob(l_nConvNum,_nID[l_nConvNum],pPick.trsf,l_nEncLatchVal)
    endIf
    //
    // Remove object from conveyor's queue
    call mot:removePart(l_nConvNum)
    //
    _nCntTransfered[l_nConvNum]=_nCntTransfered[l_nConvNum]+1
  endIf
  //
  _nID[l_nConvNum]=-1
  pPick.trsf={0,0,0,0,0,0}
  _bIsPicking=false
  //
end
